PROGRAM MAIN
VAR
	AM_Driver : AnalogMotorDriver; 
	fbSystemTime : GETSYSTEMTIME; 
	lowerHalf : UDINT; // Lower 32 bits 
	upperHalf : UDINT; // Upper 32 bits 
	fullTime : ULINT; // Combined 64 bits
	currentTimeSeconds : LREAL; 
	elapsedSeconds : LREAL; 
	
	bInitialTimeSet : BOOL := FALSE; 
	initialTimeSeconds : LREAL; // To store initial time for reference 
	
	// Output values for sine 
	rSineSignal : LREAL; 
	nPosOutputCommand : INT; 
	nNegOutputCommand : INT; 
	
END_VAR

// Poll the current system time 
fbSystemTime();
lowerHalf := fbSystemTime.timeLoDW; 
upperHalf := fbSystemTime.timeHiDW; 

fullTime := SHL(UDINT_TO_ULINT(upperHalf), 32) OR UDINT_TO_ULINT(lowerHalf); 
currentTimeSeconds := ULINT_TO_LREAL(fullTime) / 10000000.0; 

// Check to see if we need to set our initial condition. 
IF NOT bInitialTimeSet THEN
	initialTimeSeconds := currentTimeSeconds; 
	bInitialTimeSet := TRUE; 
END_IF

// Then get the DT 
elapsedSeconds := currentTimeSeconds - initialTimeSeconds; 

// Finally, pass the sine value to see what's up 
rSineSignal := 2 * SIN(elapsedSeconds * 2 * 3.14); 
AM_Driver(rCommandVoltage := rSineSignal); 
nPosOutputCommand := AM_Driver.nPosAnalogOutput; 
nNegOutputCommand := AM_Driver.nNegAnalogOutput;

END_PROGRAM

(* stored: Version 1.1.0.1, ProductVersion 3.1.4024.12
   POU MAIN: Id {60f30f80-19b9-4c10-973c-d0d6a78832e7}, SpecialFunc None *)
